PROGRAM prg_Knipperlicht
VAR
	bLamp				AT		%Q*		:BOOL;
	TimerOn: TON;
	TimerOff: TOF;
	
	//UitBreiding:
	nPotentioMeter		AT		%I*		:INT;
	Knipperfrequentie	:REAL;
	bLamp1				AT		%Q*		:BOOL;
	bLamp2				AT		%Q*		:BOOL;
	SpanningPot			AT		%Q*		:REAL;
END_VAR

//TimerOn(IN:= NOT(bLamp), PT:= T#500MS);
//TimerOff(IN:= TimerOn.Q, PT:= T#500MS, Q=> bLamp);

//Uitbreiding:
SpanningPot:= INT_TO_REAL(nPotentioMeter) * 10 / 32767;

IF (SpanningPot < 2) THEN //Frequentie 0.5Hz = 1s aan, 1s Uit
TimerOn(IN:= NOT(bLamp1), PT:= T#1S);
TimerOff(IN:= TimerOn.Q, PT:= T#1S, Q=> bLamp1);
bLamp2 := FALSE;
	ELSIF (SpanningPot >= 2) AND (SpanningPot < 4) THEN //1 Hz (500ms ON / 500ms OFF)
	TimerOn(IN:= NOT(bLamp1), PT:= T#500MS);
	TimerOff(IN:= TimerOn.Q, PT:= T#500MS, Q=> bLamp1);
	bLamp2 := FALSE;
		ELSIF (SpanningPot >= 4) AND (SpanningPot < 6) THEN //2 Hz (250ms ON / 250ms OFF)
		TimerOn(IN:= NOT(bLamp1), PT:= T#250MS);
		TimerOff(IN:= TimerOn.Q, PT:= T#250MS, Q=> bLamp1);
		bLamp2 := FALSE;
			ELSIF (SpanningPot >= 6) THEN //5Hz => 1000ms / 5 = 200ms => 200ms / 2 = 100ms AAN, 100ms UIT
			TimerOn(IN:= NOT(bLamp1), PT:= T#100MS);
			TimerOff(IN:= TimerOn.Q, PT:= T#100MS, Q=> bLamp1);
			bLamp2 := NOT(bLamp1);
END_IF

END_PROGRAM

(* stored: Version 1.1.0.1, ProductVersion 3.1.4024.15
   POU prg_Knipperlicht: Id {61454f28-08ee-4c85-9cc4-a1747181c29c}, SpecialFunc None *)
